{attribute 'linkalways'} 
{attribute 'no_explicit_call' := 'This FB is a CLASS and must be accessed using methods or properties'}
{attribute 'enable_dynamic_creation'}
FUNCTION_BLOCK Node_F_VN_DetectBlobs EXTENDS Node
VAR
    ipSrcImage : _ITcVnImage;
    ipBlobContours : _ITcVnContainer;
    stParams : _TcVnParamsBlobDetection;
    hrPrev : _HRESULT(S_OK);
	hresult : _HRESULT(S_OK);
END_VAR

METHOD PUBLIC  Clone : I_Node
VAR
	pNode : POINTER TO Node_F_VN_DetectBlobs;
END_VAR
pNode := __NEW(Node_F_VN_DetectBlobs);
Clone := pNode^;
END_METHOD

METHOD FB_init : BOOL
VAR_INPUT
	bInitRetains : BOOL; // if TRUE, the retain variables are initialized (warm start / cold start)
	bInCopyCode : BOOL;  // if TRUE, the instance afterwards gets moved into the copy code (online change)
END_VAR
AddInput('ipSrcImage', ipSrcImage);
AddInput('stParams', stParams);
AddInput('hrPrev', hrPrev);
AddOutput('ipBlobContours', ipBlobContours);
AddOutput('hresult', hresult);
END_METHOD

METHOD PROTECTED  OnExecute : HRESULT
hresult.Value := F_VN_DetectBlobs(
	ipSrcImage := ipSrcImage.Value,
    ipBlobContours := ipBlobContours.Value,
    stParams := stParams.Value,
	hrPrev:= hrPrev.Value);
END_METHOD

END_FUNCTION_BLOCK

(* stored: Version 1.1.0.1, ProductVersion 3.1.4024.13
   POU Node_F_VN_DetectBlobs: Id {50643fa5-6287-0ff7-1353-90853505476e}, SpecialFunc None
   Folder Constructor: Id {2cd9d9e8-2286-00a2-29c0-223469a37ebe}
   Method Clone: Id {95ed952e-9718-088c-1369-4d8b3370f2ee}
   Method FB_init: Id {b63a9882-1a43-0484-3b52-903fb49082a6}
   Method OnExecute: Id {0c810f61-d64b-088d-11cd-f554e6dad950} *)
